// TIA Portal V18 export
TYPE "Recipe_ShW"
// stored: IsFailsafeCompliant false
   STRUCT
      NameFeedBack : String[48];
      "Version" : Int;
      Data1 : Real;
   END_STRUCT;
END_TYPE
